PROGRAM VoltageMon
VAR
END_VAR

END_PROGRAM

(* stored: Version 1.1.0.1, ProductVersion 3.1.4024.11
   POU VoltageMon: Id {b1c07060-731f-40a5-b605-19acb84a399f}, SpecialFunc None *)
